FUNCTION_BLOCK ABSTRACT KeyValueCollectionEventHandler EXTENDS CollectionEventHandlerBase
VAR
	expectedOriginator : I_KeyValueCollection;
END_VAR

METHOD FB_init : BOOL
VAR_INPUT
	bInitRetains : BOOL; // if TRUE, the retain variables are initialized (warm start / cold start)
	bInCopyCode : BOOL;  // if TRUE, the instance afterwards gets moved into the copy code (online change)
	ExpectedOriginator : I_KeyValueCollection;
END_VAR
SetExpectedOriginator(ExpectedOriginator);
END_METHOD

METHOD PUBLIC SetExpectedOriginator
VAR_INPUT
	ExpectedOriginator : I_KeyValueCollection;
END_VAR
THIS^.expectedOriginator := ExpectedOriginator;
END_METHOD

END_FUNCTION_BLOCK

(* stored: Version 1.1.0.1, ProductVersion 3.1.4024.12
   POU KeyValueCollectionEventHandler: Id {14929a83-5297-0a9f-24b2-86e182571594}, SpecialFunc None
   Folder Constructor: Id {998ef92f-c53d-05c2-03eb-a1d8a9982a37}
   Method FB_init: Id {48178feb-cd78-0afd-069b-944a79850ae6}
   Method SetExpectedOriginator: Id {6f89679e-679b-08c4-1b0a-15e8da0e11fd} *)
